PROGRAM BrewCoffee								
VAR
	WaterTemp			:		INT;			// Water temperature 900 = 90°C
	Timer				:		TON;			// Timer for brewing the coffee

// STATES
	OFF					:		BOOL;			// Coffee machine is off
	Idle				:		BOOL;			// Waiting for input of PrepareMachine
	HeatingWater		:		BOOL;			// Water is heating up
   	BrewCoffee			: 		BOOL;			// Coffee is brewing
	State : Brewing := Brewing.OFF; 			// Current state
	
END_VAR

// Name: Jurriën Arends
// Studentnumer: 515355
// Date: 8-11-2024
// Version: 1.0

// Task 2: Brewing coffee
CASE State OF	
// STATE OFF
 Brewing.OFF:
	IF GVL.Power = FALSE THEN					// If no power, stay in this state
	  	OFF:= TRUE;
	  	Idle:= FALSE;
    END_IF
	  
    IF GVL.Power = TRUE  THEN					// IF power, go to state Idle
	  	State:= Brewing.Idle;
	  	OFF:= FALSE;

    END_IF
	
// STATE Idle 
 Brewing.Idle:
	IF GVL.Power = TRUE THEN					// If power, state is Idle
   		Idle:= TRUE;
  	END_IF
	
	IF GVL.StartBrewing = TRUE THEN				// Read variable from task 'PrepareMachine'. If machine is prepared, go to state Heating water
		State:= Brewing.HeatingWater;
		WaterTemp:= 20;							// Water temperature is 20°C
		Idle:= FALSE;
	END_IF
	
	IF GVL.Power = FALSE THEN					// If no power, go to state Off
		state:= Brewing.OFF;
		Idle:= FALSE;
	END_IF
	

// State HeatingWater
 Brewing.HeatingWater:
	IF GVL.StartBrewing = TRUE THEN				// If machine is prepared, start heating up water
	 	HeatingWater:= TRUE;
	 	WaterTemp:= WaterTemp +1;				// Add temperature + 1
	END_IF
	
	IF WaterTemp = 900 THEN						// If watertemp = 90°C (900), go to state Brew Coffee
		state:= Brewing.BrewCoffee;
		HeatingWater:= FALSE;
		GVL.StartBrewing:= FALSE;
	END_IF
	
	IF GVL.Power = FALSE THEN					// If no power, go to state Off
		state:= Brewing.OFF;
		HeatingWater:= FALSE;
	END_IF
	
// State BrewCoffee								
 Brewing.BrewCoffee:							
	IF WaterTemp = 900 THEN						// If water is heated, start brewing coffee
		BrewCoffee:= TRUE;
	END_IF
	
	Timer(IN:=TRUE, PT:=T#5S);					// Brewing time (5 sec)
	
	IF Timer.Q = TRUE THEN						// If brewing is finished, write a variable to task 'Prepare machine'. Go to state Idle
		State:=Brewing.Idle;
		BrewCoffee:= FALSE;
		Timer(IN:= FALSE);
		GVL.CoffeeBrewed:= TRUE;
	END_IF
	
	IF GVL.Power = FALSE THEN					// If no power, go to state Off
		state:= Brewing.OFF;
		BrewCoffee:= FALSE;
 	END_IF

ELSE
	OFF				:= TRUE;
	Idle			:= FALSE;
	HeatingWater	:= FALSE;
  	BrewCoffee		:= FALSE;
END_CASE;

END_PROGRAM

(* stored: Version 1.1.0.1, ProductVersion 3.1.4024.12
   POU BrewCoffee: Id {92579e20-cd9a-4b8a-a300-5b1a8846509e}, SpecialFunc None *)
